// TIA Portal project "NO & NC contacts and coils" (V16)

(* hardware
DEVICE "S7-1200 station_1"  S7-1200 Station
   slot 0: "Rack_0"  S7-1200 Rack  Rack  V1.0
   slot 1: "PLC_1"  CPU 1214C AC/DC/Rly  6ES7 214-1BG40-0XB0  V4.4
*)

// ===== PLC "PLC_1"  CPU 1214C AC/DC/Rly =====

DATA_BLOCK "entradas"   // DB1
{ S7_Optimized_Access := 'FALSE' }
VERSION : 0.1
   VAR
      entrada : Array[1..16] of Bool;
   END_VAR
BEGIN
END_DATA_BLOCK

DATA_BLOCK "salidas"   // DB2
{ S7_Optimized_Access := 'FALSE' }
VERSION : 0.1
   VAR
      salida : Array[1..16] of Bool;
   END_VAR
BEGIN
END_DATA_BLOCK

ORGANIZATION_BLOCK "Main"   // OB1, LAD, ProgramCycle
TITLE = "Main Program Sweep (Cycle)"
{ S7_Optimized_Access := 'TRUE' }
VERSION : 0.1
// Contactos y bobinas
   VAR_INPUT
      Initial_Call : Bool;   // Initial call of this OB
      Remanence : Bool;   // =True, if remanent data are available
   END_VAR
BEGIN

REGION Network 1: contactos NO y bobinas
   // **Contacto Normalmente Abierto (NO):**
   //    - Representa una condición que está **desactivada** por defecto.
   //    - Se activa (permite el paso de corriente) cuando la condición asociada es verdadera.
   //    - Símbolo: `| |`
   // 
   //    **Ejemplo:**
   //    ```
   //    | |----( )
   //    ```
   //    Cuando el contacto se cierra (verdadero), activa la bobina.
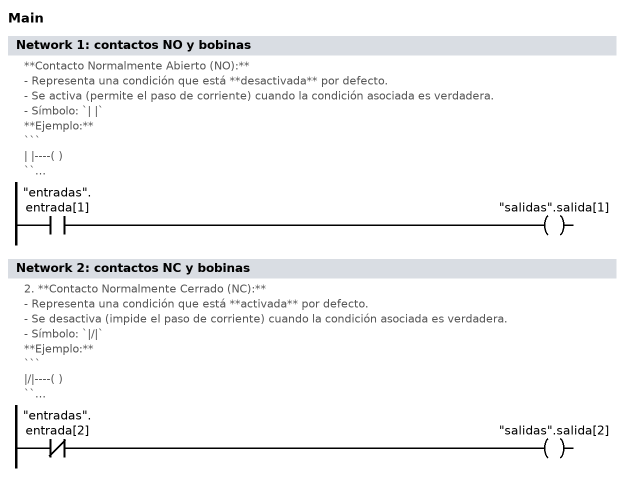
   RUNG wire#powerrail
      Contact( "entradas".entrada[1] )
      Coil( "salidas".salida[1] )
   END_RUNG
   // the same network as SCL:
   "salidas".salida[1] := "entradas".entrada[1];
END_REGION

REGION Network 2: contactos NC y bobinas
   // 2. **Contacto Normalmente Cerrado (NC):**
   //    - Representa una condición que está **activada** por defecto.
   //    - Se desactiva (impide el paso de corriente) cuando la condición asociada es verdadera.
   //    - Símbolo: `|/|`
   // 
   //    **Ejemplo:**
   //    ```
   //    |/|----( )
   //    ```
   //    El contacto interrumpe el flujo cuando se activa.
   RUNG wire#powerrail
      I_Contact( "entradas".entrada[2] )
      Coil( "salidas".salida[2] )
   END_RUNG
   // the same network as SCL:
   "salidas".salida[2] := NOT "entradas".entrada[2];
END_REGION
END_ORGANIZATION_BLOCK